TYPE ST_MonitoringAlarm :
STRUCT
    bAlarmActive: BOOL;
    bLedActive: BOOL;
    bLedAutoReset: BOOL := FALSE;
    eStatusLED: E_MonitorLed;
    eErrorLED: E_MonitorLed;
    eErrorAcknowledgeLED: E_MonitorLed;
    eEStopLED: E_MonitorLed := E_MonitorLed.eUndefined;
    eWarningLED: E_MonitorLed; //Only used for MCU400x test crates
    nErrorID: INT;
    sErrorMsg: STRING;

    //Motion Safety
    eSafetyAcknowledgeLED: E_MonitorLed;
END_STRUCT
END_TYPE

(* stored: Version 1.1.0.1
   DUT ST_MonitoringAlarm: Id {7cf4bf56-9560-4e49-afbe-1511a605e206} *)
